TYPE ST_St050_IO_IN :
STRUCT
	aFromEngelRaw	: ARRAY[0..41] OF BYTE;
	bRequestOpenProtectionDoor : BOOL;
END_STRUCT
END_TYPE

(* stored: Version 1.1.0.1
   DUT ST_St050_IO_IN: Id {cbf0f629-7aed-4e9f-95a9-262153fdd939} *)
